PROGRAM MAIN
VAR
		{attribute 'TcHmiSymbol.Show'}
	nott_cryo_ctrl : FB_NOTT_CRYO_CTRL;
END_VAR


nott_cryo_ctrl();

END_PROGRAM

(* stored: Version 1.1.0.1, ProductVersion 3.1.4026.18
   POU MAIN: Id {156d88d6-38db-460b-bb6f-1d8dbe58db4d}, SpecialFunc None *)
